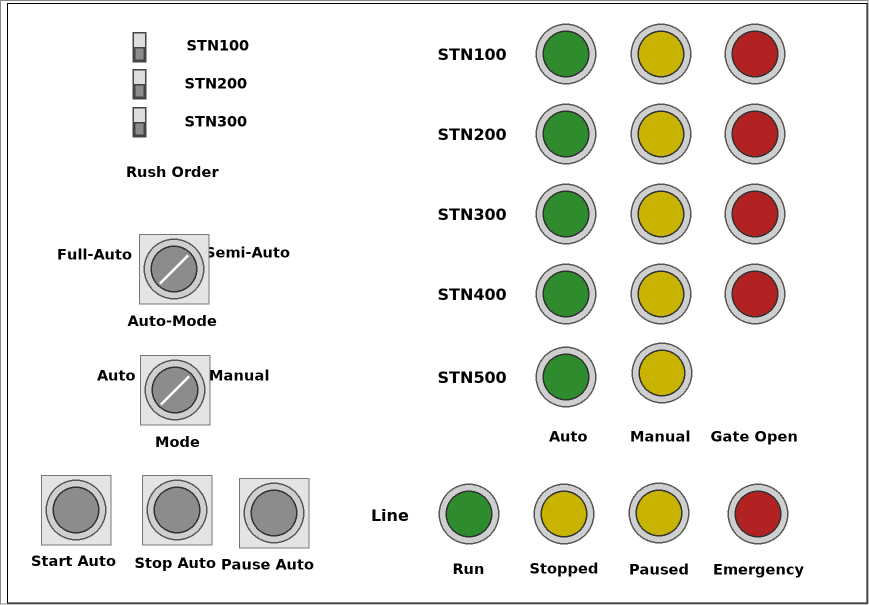
VISUALIZATION STN500HMI  // 869x605
    RoundedRectangle (7,3 860x600)
    RotarySwitch (140,355 70x70), behaviour: TOGGLE, style: Switch-RotarySwitch-Gray
    Label (93,359 47x33), "Auto"
    Label (151,427 53x30), "Mode"
    Label (203,360 73x31), "Manual"
    Label (202,239 91x27), "Semi-Auto"
    RotarySwitch (139,234 70x70), behaviour: TOGGLE, style: Switch-RotarySwitch-Gray
    Label (50,238 89x33), "Full-Auto"
    Label (121,305 103x32), "Auto-Mode"
    DipSwitch (102,107 75x30), behaviour: TOGGLE, style: Switch-DipSwitch-Gray
    DipSwitch (102,69 75x30), behaviour: TOGGLE, style: Switch-DipSwitch-Gray
    DipSwitch (102,32 75x30), behaviour: TOGGLE, style: Switch-DipSwitch-Gray
    Label (91,157 163x30), "Rush Order"
    Label (182,30 72x31), "STN100"
    Label (180,64 72x39), "STN200"
    Label (180,106 72x31), "STN300"
    Label (427,34 90x41), "STN100"
    Label (427,114 90x41), "STN200"
    Label (427,194 90x41), "STN300"
    Label (427,274 90x41), "STN400"
    Label (427,357 90x41), "STN500"
    Lamp1 (531,19 70x70), style: Lamp-Lamp1-Green
    Lamp1 (531,99 70x70), style: Lamp-Lamp1-Green
    Lamp1 (531,179 70x70), style: Lamp-Lamp1-Green
    Lamp1 (531,259 70x70), style: Lamp-Lamp1-Green
    Lamp1 (531,342 70x70), style: Lamp-Lamp1-Green
    Lamp1 (626,19 70x70), style: Lamp-Lamp1-Yellow
    Lamp1 (626,99 70x70), style: Lamp-Lamp1-Yellow
    Lamp1 (626,179 70x70), style: Lamp-Lamp1-Yellow
    Lamp1 (626,259 70x70), style: Lamp-Lamp1-Yellow
    Lamp1 (720,19 70x70), style: Lamp-Lamp1-Red
    Lamp1 (720,99 70x70), style: Lamp-Lamp1-Red
    Lamp1 (720,179 70x70), style: Lamp-Lamp1-Red
    Lamp1 (720,259 70x70), style: Lamp-Lamp1-Red
    Label (545,420 47x33), "Auto"
    Label (615,415 91x43), "Manual"
    Label (709,415 91x43), "Gate Open"
    Lamp1 (627,338 70x70), style: Lamp-Lamp1-Yellow
    PushSwitch (41,475 70x70), behaviour: TOGGLE, style: Switch-PushSwitch-Gray
    PushSwitch (142,475 70x70), behaviour: TOGGLE, style: Switch-PushSwitch-Gray
    PushSwitch (239,478 70x70), behaviour: TOGGLE, style: Switch-PushSwitch-Gray
    Label (31,544 85x34), "Start Auto"
    Label (133,546 85x34), "Stop Auto"
    Label (219,546 97x37), "Pause Auto"
    Label (345,495 90x41), "Line"
    Lamp1 (434,479 70x70), style: Lamp-Lamp1-Green
    Lamp1 (529,479 70x70), style: Lamp-Lamp1-Yellow
    Lamp1 (723,479 70x70), style: Lamp-Lamp1-Red
    Label (713,548 91x43), "Emergency"
    Lamp1 (624,478 70x70), style: Lamp-Lamp1-Yellow
    Label (442,554 53x30), "Run"
    Label (523,555 82x27), "Stopped"
    Label (618,556 82x27), "Paused"
END_VISUALIZATION

(* stored: Version 1.1.0.1, ProductVersion 3.1.4024.2
   Visu STN500HMI: Id {b2985b79-7953-4416-af03-59971a9eb832} *)
